// TIA Portal V19 export
VAR_GLOBAL   // PLC tag table "conveyor6m"
   "Belt Conveyor (6m) 0" AT %Q0.4 : Bool;
END_VAR
